(* Logix 5000 project; controller cal1632 1756-L62 rev 16.20; software revision 16.05; part 57 of 57 *)
(* tags used below, declared in another part *)
   AFI : BOOL;
   FAULT : BOOL;
   HMI : BOOL;
   p01r09 : routine;
   p01r09_pb_global_reset : BOOL;
   p30_di_pin_1 : BOOL;
   p30_di_pin_2 : BOOL;
   p30_di_pin_3 : BOOL;
   p30_di_pin_4 : BOOL;
   p30_di_pin_5 : BOOL;
   p30_di_pin_6 : BOOL;
   p30_di_pin_7 : BOOL;
   p30_di_pin_8 : BOOL;
   p30_di_retraction_down_ls : BOOL;
   p30_di_retraction_up_ls : BOOL;
   p30_di_rotation_fault : BOOL;
   p30_di_ss_close : BOOL;
   p30_di_ss_open : BOOL;
   p30_dint_to_hmi : DINT[16];
   p30_do_retract_motion : BOOL;
   p30_do_rotation_fwd : BOOL;
   p30_do_rotation_rev : BOOL;
   p30r08 : routine;
   p30r08_timer_fault : TIMER[4];
   p30r08_timer_warning : TIMER[4];
   p30r09 : routine;
   p30r09_mode_close : BOOL;
   p30r09_mode_off : BOOL;
   p30r09_mode_open : BOOL;
   p30r09_timer_fault : TIMER[4];
   p30r09_timer_warning : TIMER[4];
   p30r10 : routine;
   p30r10_motion_monitor_dwell : TIMER;
   p30r10_request_close : BOOL;
   p30r10_request_monitor : BOOL;
   p30r10_request_open : BOOL;
   p30r10_run_permissive : BOOL;
   p30r10_safety_pins_stowed : BOOL;
   p30r10_timer_fault : TIMER[4];
   p30r10_timer_warning : TIMER[4];
(* P30_Retraction_System, continued *)

ROUTINE R08_Warnings   (* ladder *)
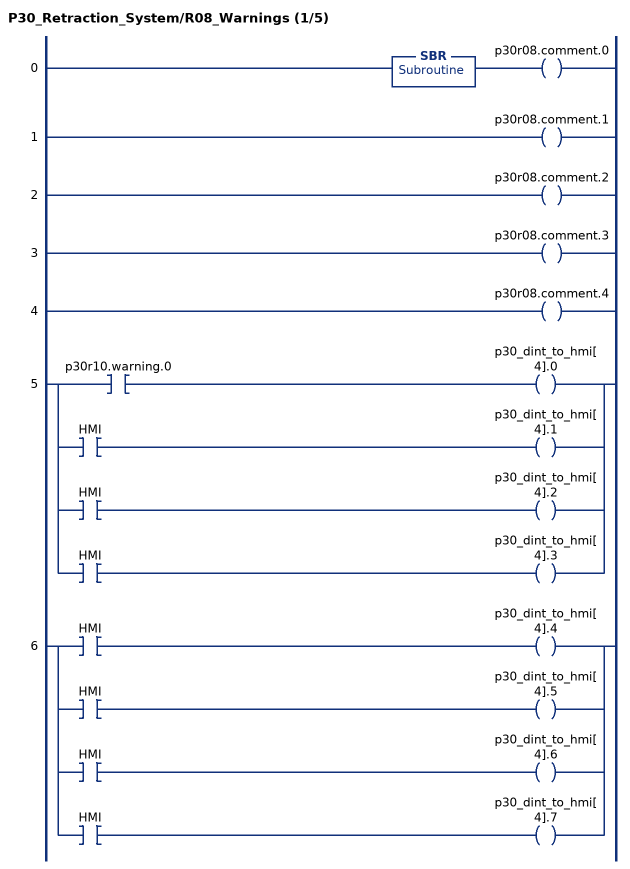
   0: SBR()OTE(p30r08.comment.0);
   1: OTE(p30r08.comment.1);
   2: OTE(p30r08.comment.2);
   3: OTE(p30r08.comment.3);
   4: OTE(p30r08.comment.4);
   5: [XIC(p30r10.warning.0) OTE(p30_dint_to_hmi[4].0) ,XIC(HMI) OTE(p30_dint_to_hmi[4].1) ,XIC(HMI) OTE(p30_dint_to_hmi[4].2) ,XIC(HMI) OTE(p30_dint_to_hmi[4].3) ];
   6: [XIC(HMI) OTE(p30_dint_to_hmi[4].4) ,XIC(HMI) OTE(p30_dint_to_hmi[4].5) ,XIC(HMI) OTE(p30_dint_to_hmi[4].6) ,XIC(HMI) OTE(p30_dint_to_hmi[4].7) ];
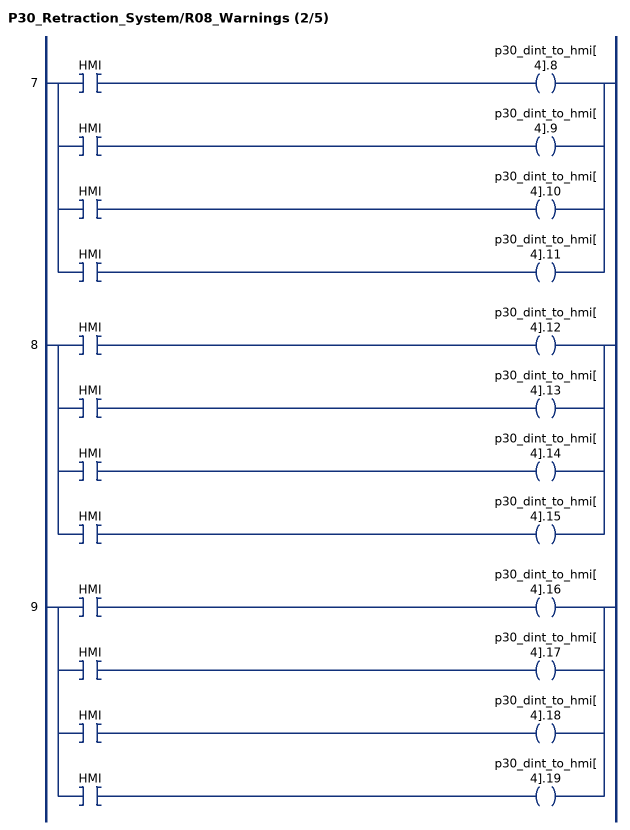
   7: [XIC(HMI) OTE(p30_dint_to_hmi[4].8) ,XIC(HMI) OTE(p30_dint_to_hmi[4].9) ,XIC(HMI) OTE(p30_dint_to_hmi[4].10) ,XIC(HMI) OTE(p30_dint_to_hmi[4].11) ];
   8: [XIC(HMI) OTE(p30_dint_to_hmi[4].12) ,XIC(HMI) OTE(p30_dint_to_hmi[4].13) ,XIC(HMI) OTE(p30_dint_to_hmi[4].14) ,XIC(HMI) OTE(p30_dint_to_hmi[4].15) ];
   9: [XIC(HMI) OTE(p30_dint_to_hmi[4].16) ,XIC(HMI) OTE(p30_dint_to_hmi[4].17) ,XIC(HMI) OTE(p30_dint_to_hmi[4].18) ,XIC(HMI) OTE(p30_dint_to_hmi[4].19) ];
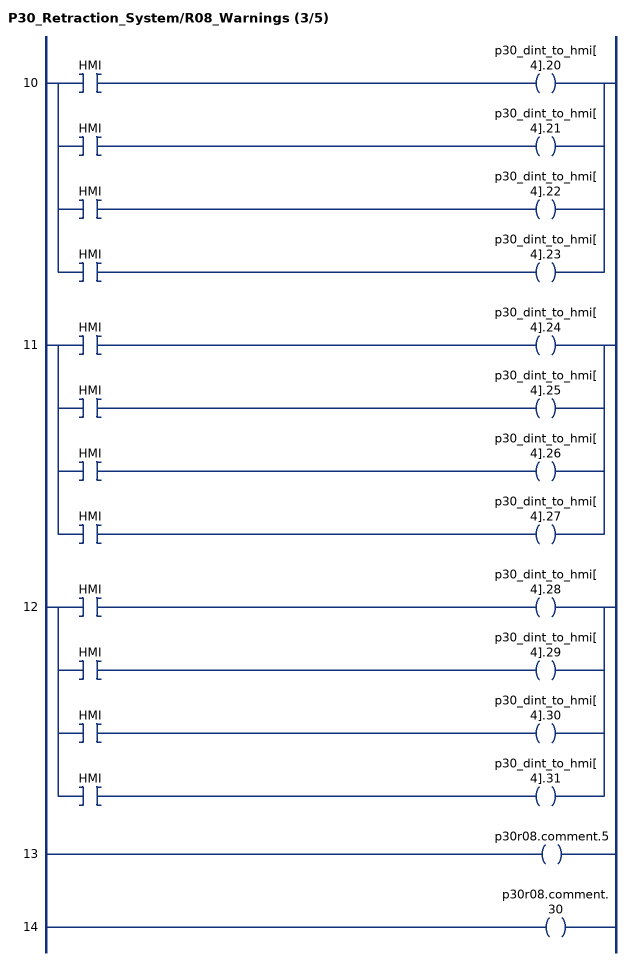
   10: [XIC(HMI) OTE(p30_dint_to_hmi[4].20) ,XIC(HMI) OTE(p30_dint_to_hmi[4].21) ,XIC(HMI) OTE(p30_dint_to_hmi[4].22) ,XIC(HMI) OTE(p30_dint_to_hmi[4].23) ];
   11: [XIC(HMI) OTE(p30_dint_to_hmi[4].24) ,XIC(HMI) OTE(p30_dint_to_hmi[4].25) ,XIC(HMI) OTE(p30_dint_to_hmi[4].26) ,XIC(HMI) OTE(p30_dint_to_hmi[4].27) ];
   12: [XIC(HMI) OTE(p30_dint_to_hmi[4].28) ,XIC(HMI) OTE(p30_dint_to_hmi[4].29) ,XIC(HMI) OTE(p30_dint_to_hmi[4].30) ,XIC(HMI) OTE(p30_dint_to_hmi[4].31) ];
   13: OTE(p30r08.comment.5);
   14: OTE(p30r08.comment.30);
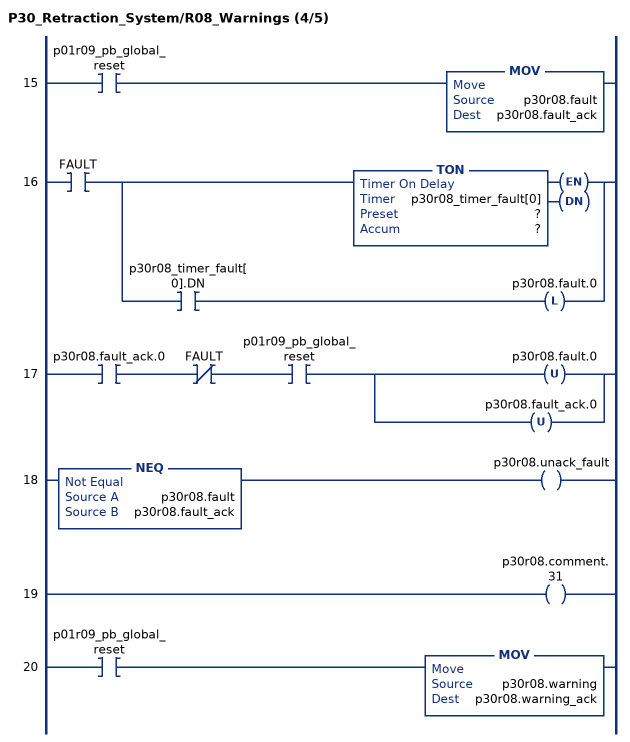
   15: XIC(p01r09_pb_global_reset)MOV(p30r08.fault,p30r08.fault_ack);
   16: XIC(FAULT)[TON(p30r08_timer_fault[0],?,?) ,XIC(p30r08_timer_fault[0].DN) OTL(p30r08.fault.0) ];
   17: XIC(p30r08.fault_ack.0)XIO(FAULT)XIC(p01r09_pb_global_reset)[OTU(p30r08.fault.0) ,OTU(p30r08.fault_ack.0) ];
   18: NEQ(p30r08.fault,p30r08.fault_ack)OTE(p30r08.unack_fault);
   19: OTE(p30r08.comment.31);
   20: XIC(p01r09_pb_global_reset)MOV(p30r08.warning,p30r08.warning_ack);
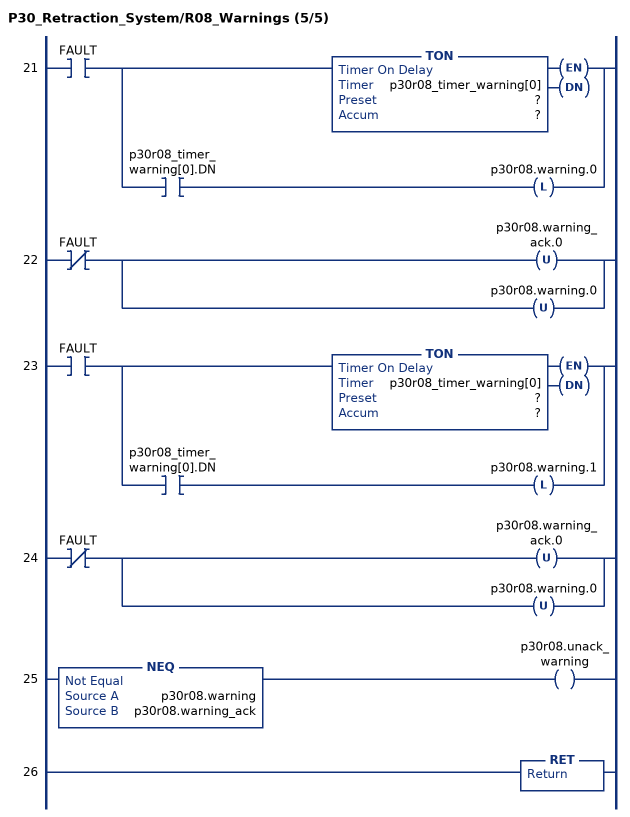
   21: XIC(FAULT)[TON(p30r08_timer_warning[0],?,?) ,XIC(p30r08_timer_warning[0].DN) OTL(p30r08.warning.0) ];
   22: XIO(FAULT)[OTU(p30r08.warning_ack.0) ,OTU(p30r08.warning.0) ];
   23: XIC(FAULT)[TON(p30r08_timer_warning[0],?,?) ,XIC(p30r08_timer_warning[0].DN) OTL(p30r08.warning.1) ];
   24: XIO(FAULT)[OTU(p30r08.warning_ack.0) ,OTU(p30r08.warning.0) ];
   25: NEQ(p30r08.warning,p30r08.warning_ack)OTE(p30r08.unack_warning);
   26: RET();
END_ROUTINE

ROUTINE R09_Modes   (* ladder *)
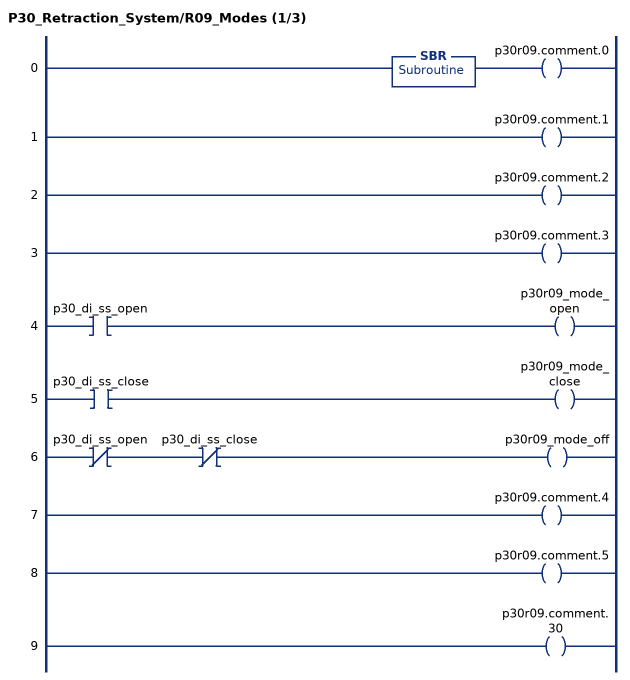
   0: SBR()OTE(p30r09.comment.0);
   1: OTE(p30r09.comment.1);
   2: OTE(p30r09.comment.2);
   3: OTE(p30r09.comment.3);
   4: XIC(p30_di_ss_open)OTE(p30r09_mode_open);
   5: XIC(p30_di_ss_close)OTE(p30r09_mode_close);
   6: XIO(p30_di_ss_open)XIO(p30_di_ss_close)OTE(p30r09_mode_off);
   7: OTE(p30r09.comment.4);
   8: OTE(p30r09.comment.5);
   9: OTE(p30r09.comment.30);
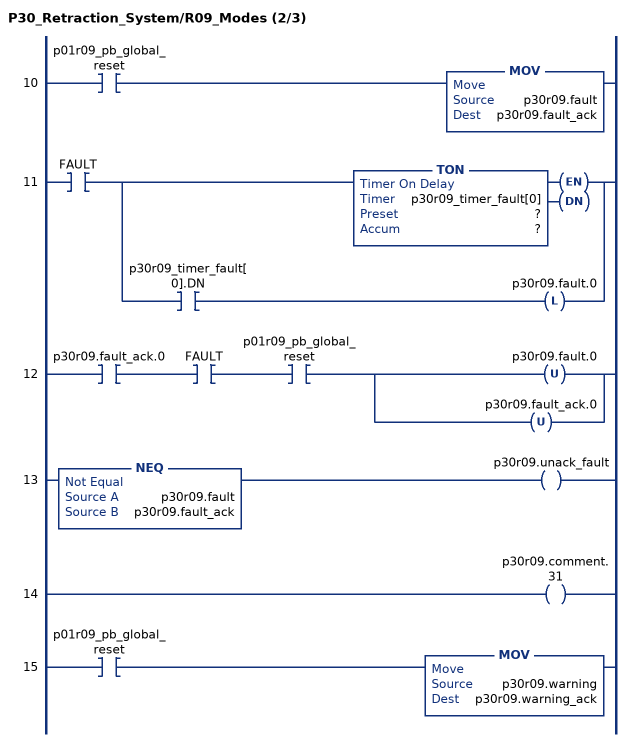
   10: XIC(p01r09_pb_global_reset)MOV(p30r09.fault,p30r09.fault_ack);
   11: XIC(FAULT)[TON(p30r09_timer_fault[0],?,?) ,XIC(p30r09_timer_fault[0].DN) OTL(p30r09.fault.0) ];
   12: XIC(p30r09.fault_ack.0)XIC(FAULT)XIC(p01r09_pb_global_reset)[OTU(p30r09.fault.0) ,OTU(p30r09.fault_ack.0) ];
   13: NEQ(p30r09.fault,p30r09.fault_ack)OTE(p30r09.unack_fault);
   14: OTE(p30r09.comment.31);
   15: XIC(p01r09_pb_global_reset)MOV(p30r09.warning,p30r09.warning_ack);
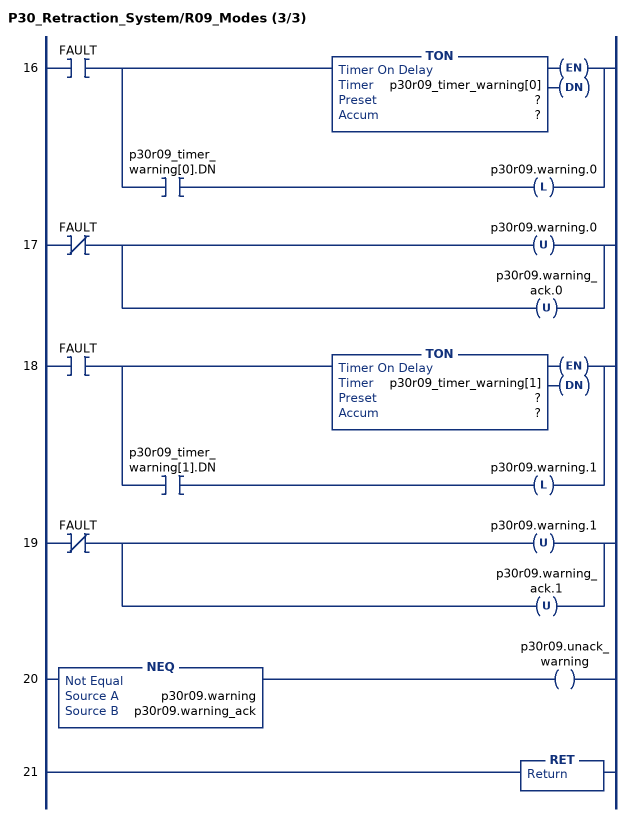
   16: XIC(FAULT)[TON(p30r09_timer_warning[0],?,?) ,XIC(p30r09_timer_warning[0].DN) OTL(p30r09.warning.0) ];
   17: XIO(FAULT)[OTU(p30r09.warning.0) ,OTU(p30r09.warning_ack.0) ];
   18: XIC(FAULT)[TON(p30r09_timer_warning[1],?,?) ,XIC(p30r09_timer_warning[1].DN) OTL(p30r09.warning.1) ];
   19: XIO(FAULT)[OTU(p30r09.warning.1) ,OTU(p30r09.warning_ack.1) ];
   20: NEQ(p30r09.warning,p30r09.warning_ack)OTE(p30r09.unack_warning);
   21: RET();
END_ROUTINE

ROUTINE R10_Retraction   (* ladder *)
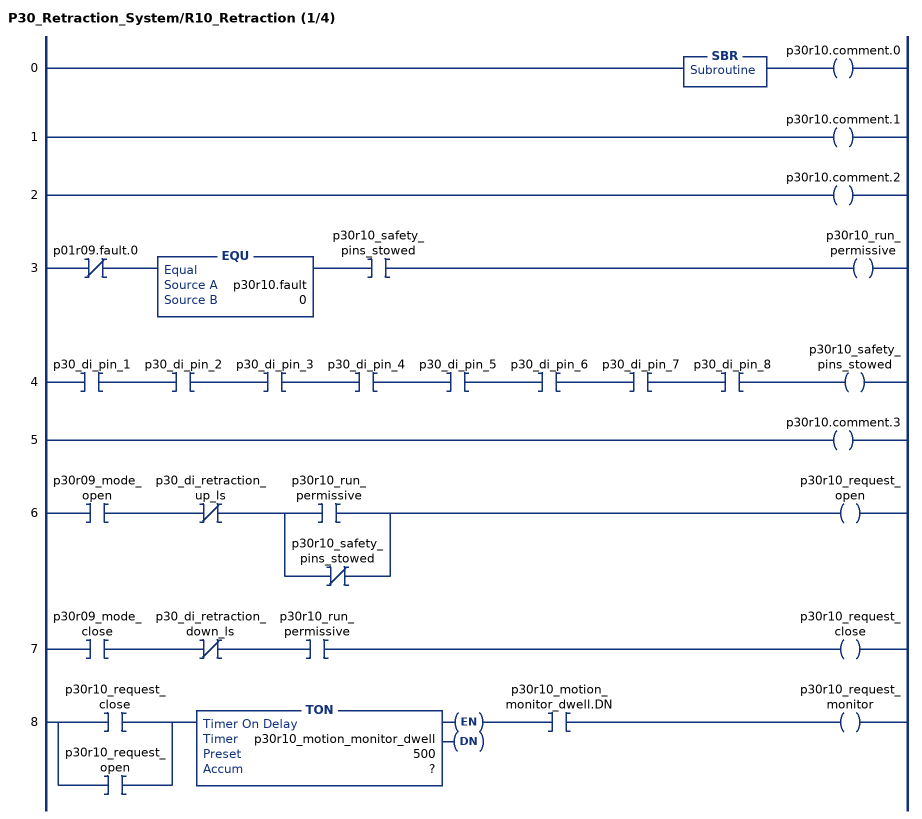
   0: SBR()OTE(p30r10.comment.0);
   1: OTE(p30r10.comment.1);
   2: OTE(p30r10.comment.2);
   3: XIO(p01r09.fault.0)EQU(p30r10.fault,0)XIC(p30r10_safety_pins_stowed)OTE(p30r10_run_permissive);
   4: XIC(p30_di_pin_1)XIC(p30_di_pin_2)XIC(p30_di_pin_3)XIC(p30_di_pin_4)XIC(p30_di_pin_5)XIC(p30_di_pin_6)XIC(p30_di_pin_7)XIC(p30_di_pin_8)OTE(p30r10_safety_pins_stowed);
   5: OTE(p30r10.comment.3);
   6: XIC(p30r09_mode_open)XIO(p30_di_retraction_up_ls)[XIC(p30r10_run_permissive) ,XIO(p30r10_safety_pins_stowed) ]OTE(p30r10_request_open);
   7: XIC(p30r09_mode_close)XIO(p30_di_retraction_down_ls)XIC(p30r10_run_permissive)OTE(p30r10_request_close);
   8: [XIC(p30r10_request_close) ,XIC(p30r10_request_open) ]TON(p30r10_motion_monitor_dwell,?,?)XIC(p30r10_motion_monitor_dwell.DN)OTE(p30r10_request_monitor);
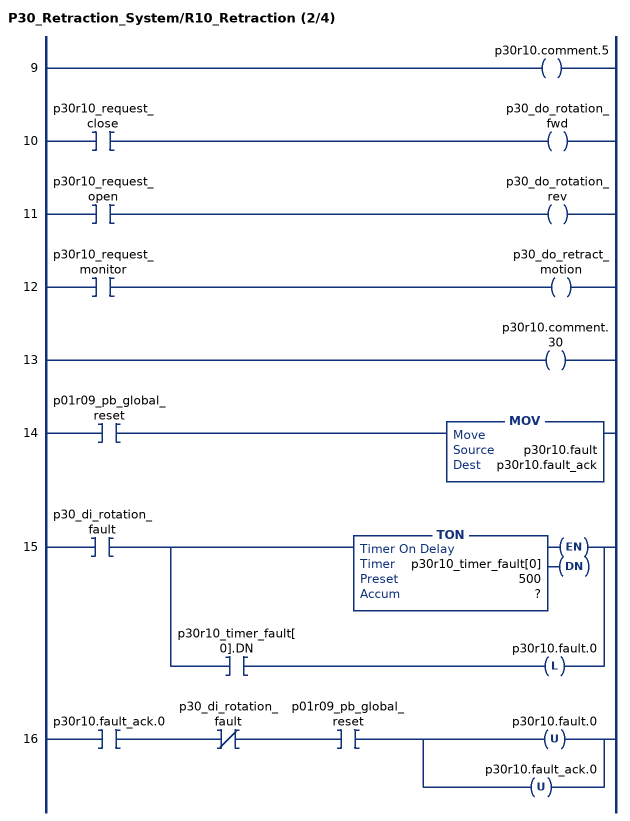
   9: OTE(p30r10.comment.5);
   10: XIC(p30r10_request_close)OTE(p30_do_rotation_fwd);
   11: XIC(p30r10_request_open)OTE(p30_do_rotation_rev);
   12: XIC(p30r10_request_monitor)OTE(p30_do_retract_motion);
   13: OTE(p30r10.comment.30);
   14: XIC(p01r09_pb_global_reset)MOV(p30r10.fault,p30r10.fault_ack);
   15: XIC(p30_di_rotation_fault)[TON(p30r10_timer_fault[0],?,?) ,XIC(p30r10_timer_fault[0].DN) OTL(p30r10.fault.0) ];
   16: XIC(p30r10.fault_ack.0)XIO(p30_di_rotation_fault)XIC(p01r09_pb_global_reset)[OTU(p30r10.fault.0) ,OTU(p30r10.fault_ack.0) ];
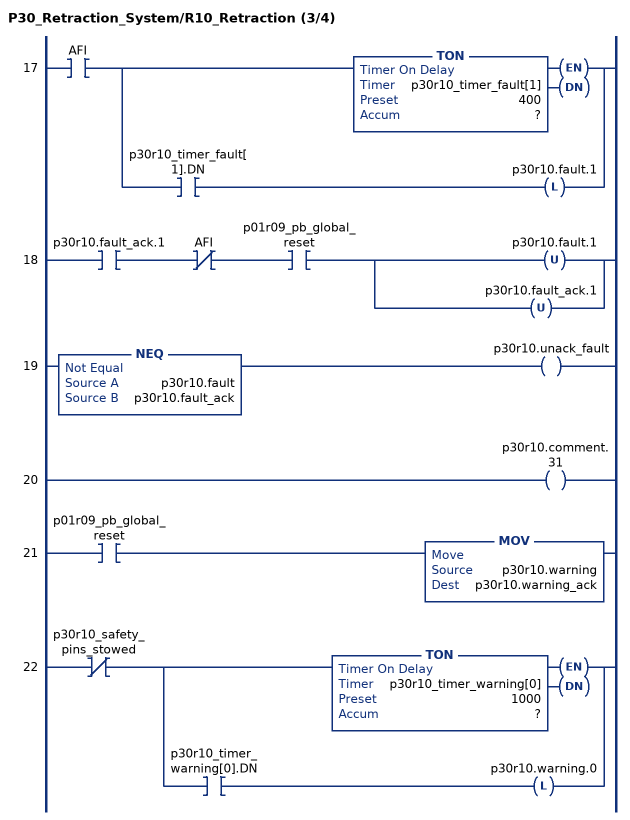
   17: XIC(AFI)[TON(p30r10_timer_fault[1],?,?) ,XIC(p30r10_timer_fault[1].DN) OTL(p30r10.fault.1) ];
   18: XIC(p30r10.fault_ack.1)XIO(AFI)XIC(p01r09_pb_global_reset)[OTU(p30r10.fault.1) ,OTU(p30r10.fault_ack.1) ];
   19: NEQ(p30r10.fault,p30r10.fault_ack)OTE(p30r10.unack_fault);
   20: OTE(p30r10.comment.31);
   21: XIC(p01r09_pb_global_reset)MOV(p30r10.warning,p30r10.warning_ack);
   22: XIO(p30r10_safety_pins_stowed)[TON(p30r10_timer_warning[0],?,?) ,XIC(p30r10_timer_warning[0].DN) OTL(p30r10.warning.0) ];
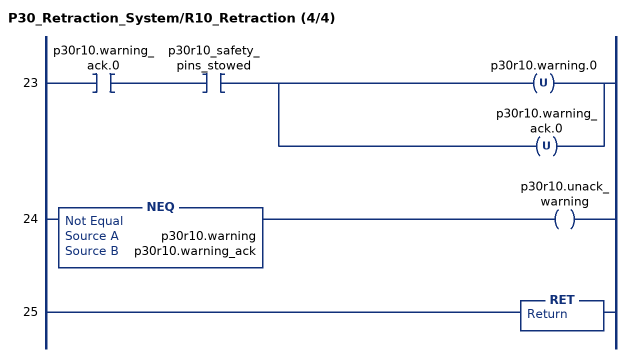
   23: XIC(p30r10.warning_ack.0)XIC(p30r10_safety_pins_stowed)[OTU(p30r10.warning.0) ,OTU(p30r10.warning_ack.0) ];
   24: NEQ(p30r10.warning,p30r10.warning_ack)OTE(p30r10.unack_warning);
   25: RET();
END_ROUTINE
END_PROGRAM
